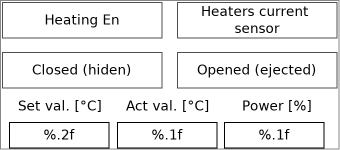
VISUALIZATION vHP3_HeatedPlateMain  // 340x150
VAR_IN_OUT
	fbHP	: fbHPv3_Control;
END_VAR
    Rectangle (9,122 100x26), "%.2f", text variable: fbHP.fbHP_PID.SET_POINT
    Label (10,93 100x26), "Set val. [°C]"
    Rectangle (117,122 100x26), "%.1f", text variable: fbHP.fbHP_PID.ACTUAL
    Label (118,93 100x26), "Act val. [°C]"
    Rectangle (224,122 100x26), "%.1f", text variable: fbHP.rHPHeaterPower, colour toggle: fbHP.rHPHeaterPower > 90.0
    Label (225,93 104x26), "Power [%]"
    Rectangle (177,2 160x36), "Heaters current sensor", colour toggle: fbHP.stInOuts.bI_HeaterCurrentSensor
    Rectangle (2,2 160x36), "Heating En", colour toggle: fbHP.fbHP_HeaterON.Q
    Rectangle (2,52 160x36), "Closed (hiden)", colour toggle: fbHP.fbHeatedPlate_Actuator.Closed
    Rectangle (177,52 160x36), "Opened (ejected)", colour toggle: fbHP.fbHeatedPlate_Actuator.Opened
END_VISUALIZATION

(* stored: Version 1.1.0.1, ProductVersion 3.1.4024.12
   Visu vHP3_HeatedPlateMain: Id {b3d2d2ac-9644-4a5c-ba61-cbf790eb765f} *)
